// SIMATIC S7-200 project (STEP 7-Micro/WIN), CPU 226 REL 02.01

ORGANIZATION_BLOCK MAIN:OB1
TITLE=PROGRAM COMMENTS
BEGIN
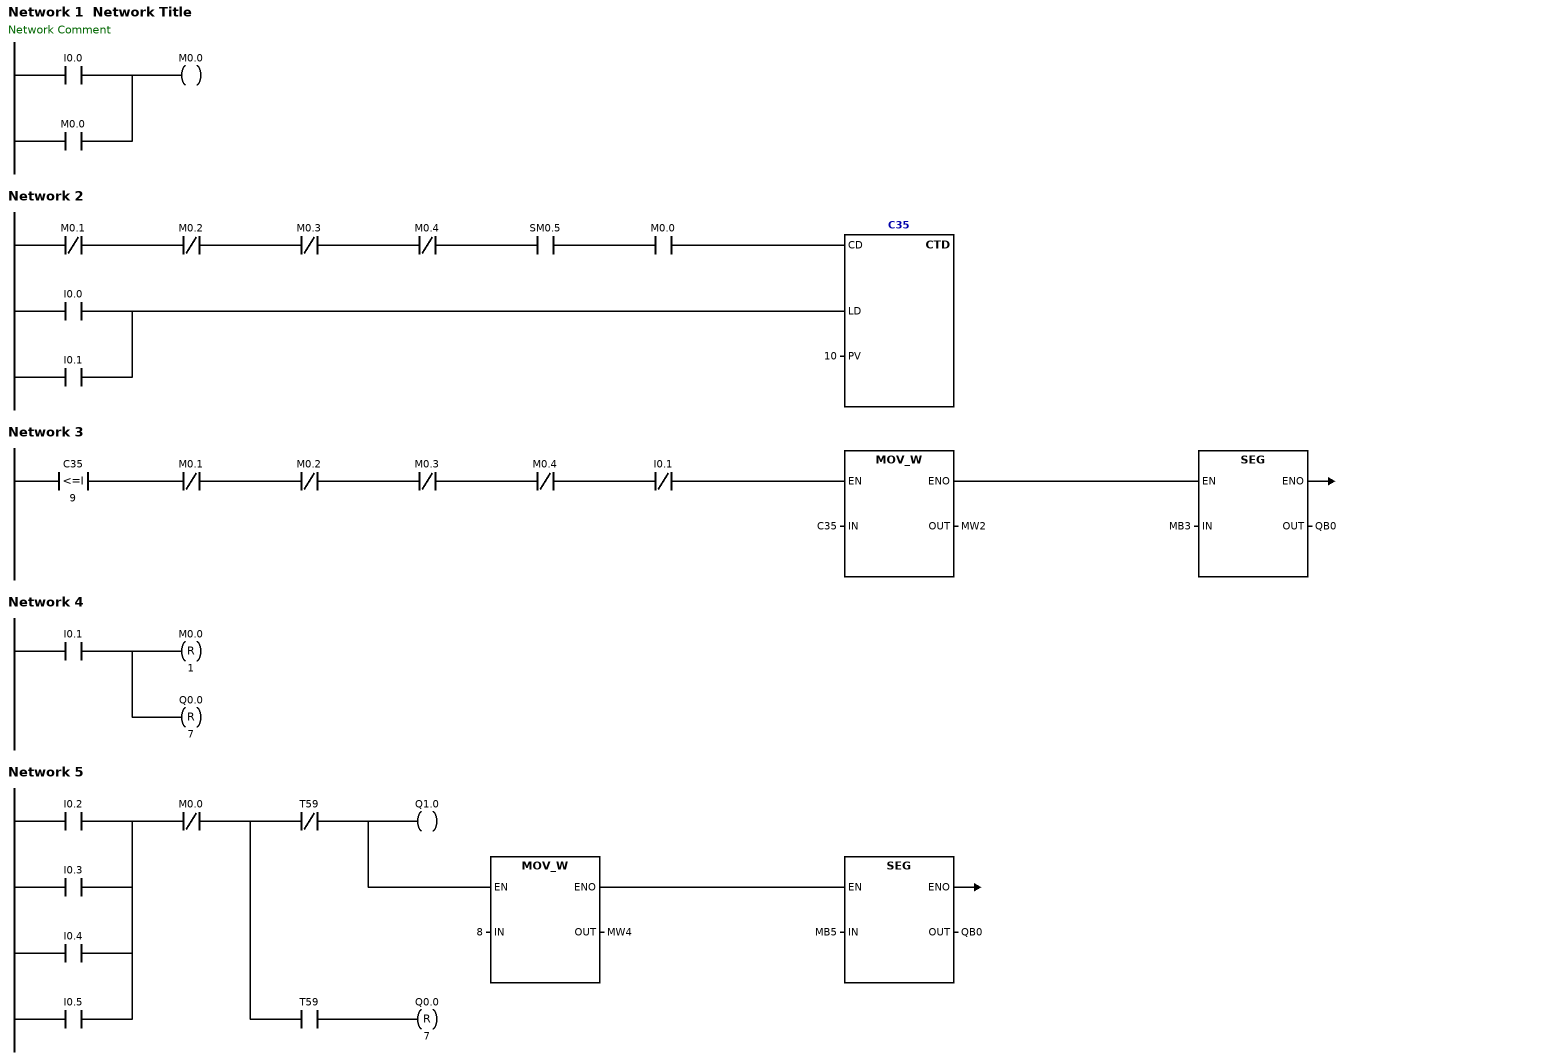
Network 1 // Network Title
// Network Comment
LD     I0.0
O      M0.0
=      M0.0
Network 2
LDN    M0.1
AN     M0.2
AN     M0.3
AN     M0.4
A      SM0.5
A      M0.0
LD     I0.0
O      I0.1
CTD    C35, 10
Network 3
LDW<=  C35, 9
AN     M0.1
AN     M0.2
AN     M0.3
AN     M0.4
AN     I0.1
MOVW   C35, MW2
AENO
SEG    MB3, QB0
Network 4
LD     I0.1
R      M0.0, 1
R      Q0.0, 7
Network 5
LD     I0.2
O      I0.3
O      I0.4
O      I0.5
AN     M0.0
LPS
AN     T59
=      Q1.0
MOVW   8, MW4
AENO
SEG    MB5, QB0
LPP
A      T59
R      Q0.0, 7
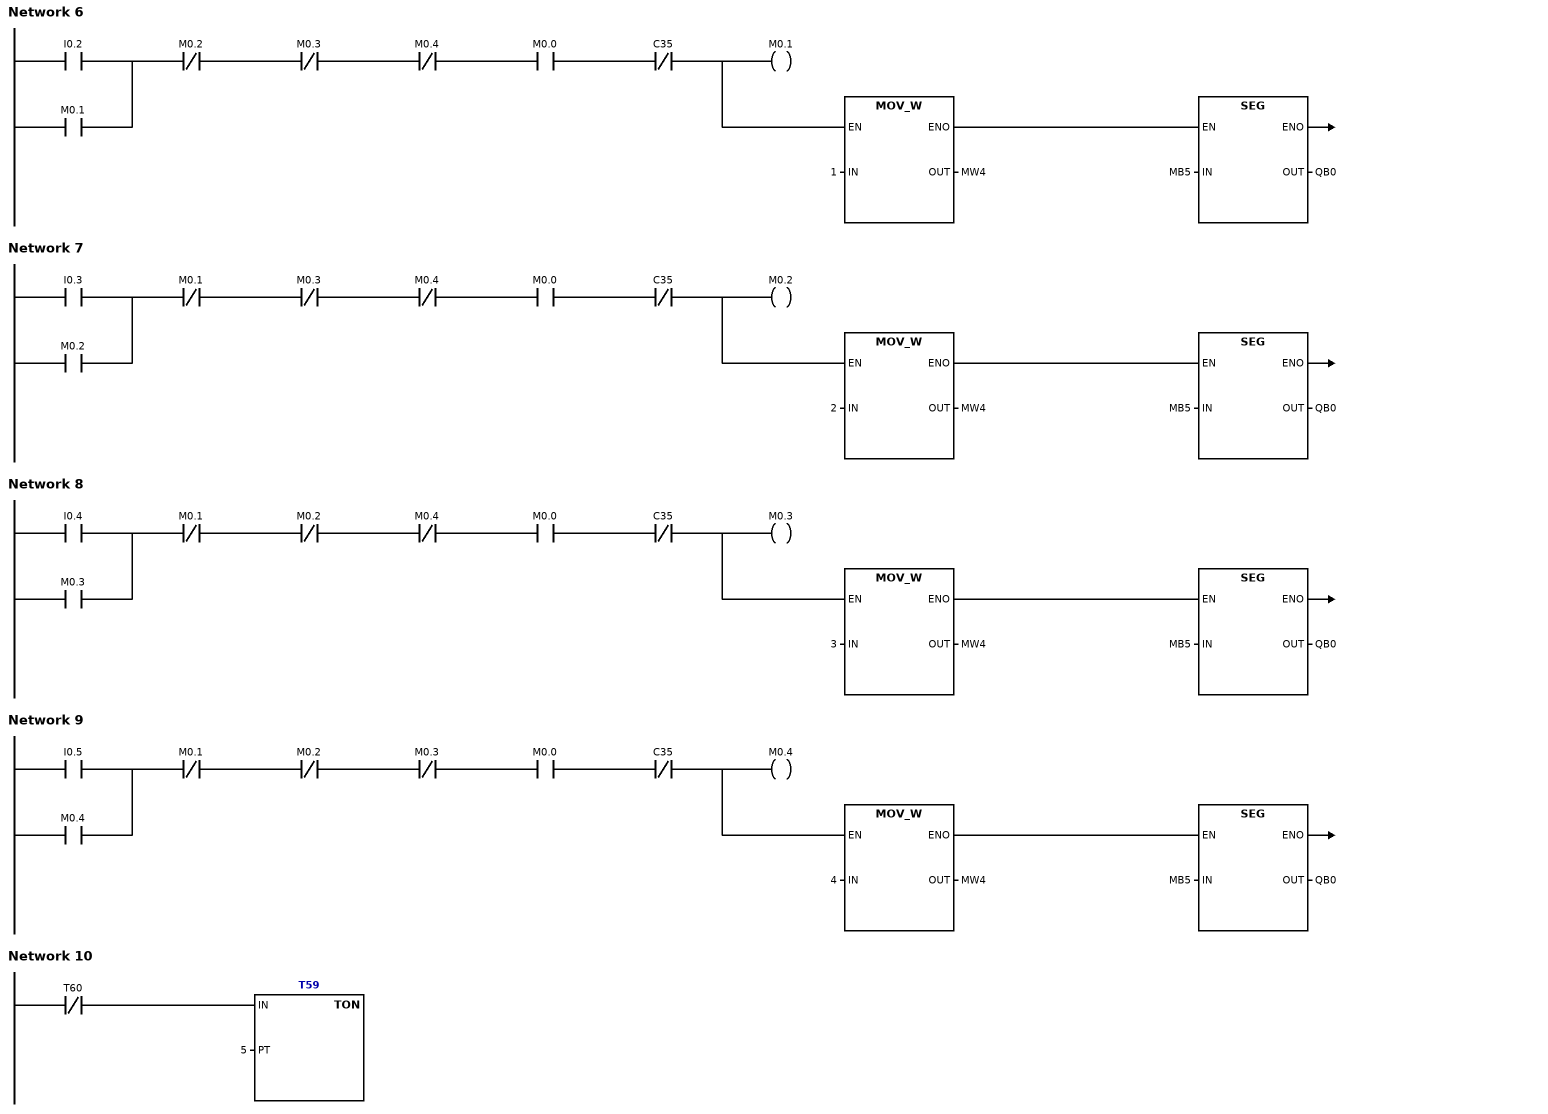
Network 6
LD     I0.2
O      M0.1
AN     M0.2
AN     M0.3
AN     M0.4
A      M0.0
AN     C35
=      M0.1
MOVW   1, MW4
AENO
SEG    MB5, QB0
Network 7
LD     I0.3
O      M0.2
AN     M0.1
AN     M0.3
AN     M0.4
A      M0.0
AN     C35
=      M0.2
MOVW   2, MW4
AENO
SEG    MB5, QB0
Network 8
LD     I0.4
O      M0.3
AN     M0.1
AN     M0.2
AN     M0.4
A      M0.0
AN     C35
=      M0.3
MOVW   3, MW4
AENO
SEG    MB5, QB0
Network 9
LD     I0.5
O      M0.4
AN     M0.1
AN     M0.2
AN     M0.3
A      M0.0
AN     C35
=      M0.4
MOVW   4, MW4
AENO
SEG    MB5, QB0
Network 10
LDN    T60
TON    T59, 5
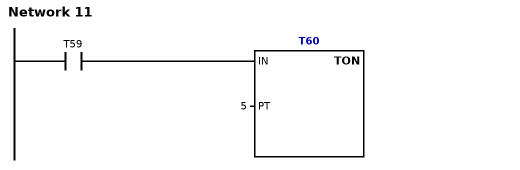
Network 11
LD     T59
TON    T60, 5
END_ORGANIZATION_BLOCK
